FUNCTION_BLOCK F_WSTRING_AS_BYTE (* Convert WSTRING to BYTE *)
  (* Standard: 61499-1; Description: Copyright (c) 2023 Martin Erich Jobst This program and the accompanying materials are made available under the terms of the Eclipse Public License 2.0 which is available at https://www.eclipse.org/legal/epl-2.0/ SPDX-License-Identifier: EPL-2.0 *)
  (* Version 3.0, 2025-04-14, Patrick Aigner, changed package *)
  (* Version 1.0, 2023-04-28, Martin Jobst *)
  PACKAGE iec61131::conversion;
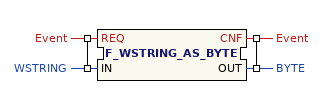
  EVENT_INPUT
    REQ WITH IN; (* Normal Execution Request *)
  END_EVENT
  EVENT_OUTPUT
    CNF WITH OUT; (* Execution Confirmation *)
  END_EVENT
  VAR_INPUT
    IN : WSTRING;
  END_VAR
  VAR_OUTPUT
    OUT : BYTE;
  END_VAR
  EC_STATES
    REQ : REQ -> CNF;
  END_STATES
  ALGORITHM REQ IN ST:
OUT := WSTRING_AS_BYTE(IN);
  END_ALGORITHM
END_FUNCTION_BLOCK
